Yaskawa INFORM job: USER_FRAME_50_CALC.JBI

/JOB
//NAME USER_FRAME_50_CALC
//POS
///NPOS 1,1,0,3,3,0
///USER 50
///TOOL 0
///POSTYPE USER
///RECTAN
///RCONF 0,0,1,0,0,0,0,0,0,0,0,0,0,0,0,0,0,0,0,0,0,0,0,0
C00000=5303.253,22.899,150.358,-0.0446,-75.9700,0.0375
///RCONF 0,0,0,0,0,0,0,0,0,0,0,0,0,0,0,0,0,0,0,0,0,0,0,0
BC00000=3342.174
///POSTYPE BASE
P00007=-200.000,0.000,0.000,0.0000,0.0000,0.0000
P00008=5000.000,0.000,0.000,0.0000,0.0000,0.0000
P00009=0.000,5000.000,0.000,0.0000,0.0000,0.0000
BP00007=-200.000
BP00008=0.000
BP00009=0.000
//INST
///DATE 2024/10/24 12:09
///ATTR SC,RW,RJ
////FRAME USER 50
///GROUP1 RB1,BS1
///LVARS 0,0,1,0,0,0,0,0
NOP
'*
'*
'*
'PROGRAM DO PRZESUWANIA POZYCJI
'RAMY PRZEDNIEJ
'WYKORZYSTUJACY SYGNALY Z KONIKA
'*
'*
'*
SUB LD000 LD000
'5040 WARTOSC -300
IFTHENEXP IN#(1737)=ON
	 SET LD000 -300
ENDIF
'5140 WARTOSC -200
IFTHENEXP IN#(1738)=ON
	 SET LD000 -200
ENDIF
'5240 WARTOSC -100
IFTHENEXP IN#(1739)=ON
	 SET LD000 -100
ENDIF
'5340 UKLAD BAZOWY WARTOSC 0
IFTHENEXP IN#(1740)=ON
	 SET LD000 0
ENDIF
'5440 WARTOSC 100
IFTHENEXP IN#(1741)=ON
	 SET LD000 100
ENDIF
IFTHENEXP LD000>1000 OREXP LD000<-1000
	 SETUALM 8555 S005 0
ENDIF
MUL LD000 1000
SETE P0007 (1) LD000
SETE P0007 (2) 0
SETE P0007 (3) 0
SETE P0007 (4) 0
SETE P0007 (5) 0
SETE P0007 (6) 0
SETE BP007 (1) LD000
SETE BP007 (2) 0
SETE BP007 (3) 0
SETE BP007 (4) 0
SETE BP007 (5) 0
SETE BP007 (6) 0
SETE P0008 (1) 5000000
SETE P0008 (2) 0
SETE P0008 (3) 0
SETE P0008 (4) 0
SETE P0008 (5) 0
SETE P0008 (6) 0
SETE BP008 (1) 0
SETE BP008 (2) 0
SETE BP008 (3) 0
SETE BP008 (4) 0
SETE BP008 (5) 0
SETE BP008 (6) 0
SETE P0009 (1) 0
SETE P0009 (2) 5000000
SETE P0009 (3) 0
SETE P0009 (4) 0
SETE P0009 (5) 0
SETE P0009 (6) 0
SETE BP009 (1) 0
SETE BP009 (2) 0
SETE BP009 (3) 0
SETE BP009 (4) 0
SETE BP009 (5) 0
SETE BP009 (6) 0
MFRAME UF#(50) PX0007 PX0008 PX0009
MOVJ C00000 BC00000 VJ=50.00
END
